# EPICS StreamDevice protocol: visarCameraApp/srcProtocol/visar.proto
################################################
#                                              #
#  Stream Protocol File for the Visar camera   #
#                                              #
#                                              #
################################################

OutTerminator =  CR;
ReplyTimeout  =  300;
ReadTimeout   =  100;
WriteTimeout  =  100;
LockTimeout   =  300;

###############################################
#  Camera Parameters                          #
###############################################

#########################################
#  Exposure time                        #
#########################################

set_exposure_time{
    InTerminator = ;
    ExtraInput   = Ignore;
	out "CamParamSet(Live,Exposure,%.6f %(\$1AcquireTimeVisarUnits){us|ms|s|min})";
	in "%*/(?m)0,CamParamSet\r/";
}

set_exposure_time_s{
    InTerminator = ;
    ExtraInput   = Ignore;
	out "CamParamSet(Live,Exposure,%(\$1AcquireTime).6f s)";
	in "%*/(?m)0,CamParamSet\r/";
}

get_exposure_time{
    InTerminator = ;
    ExtraInput   = Ignore;
	out "CamParamGet(Live,Exposure)";
	in  "%*/(?m)0,CamParamGet,/%f %(\$1AcquireTimeVisarUnits_RBV){us|ms|s|m}\r";
}

#########################################
#  Gain                                 #
#########################################

# II Gain / AD Gain
set_II_gain{
    InTerminator = ;
    ExtraInput   = Ignore;
	out "DevParamSet(TD,II-Gain,%d)";
	in "%*/(?m)0,DevParamSet\r/";
}

get_II_gain{
    InTerminator = "";
    ExtraInput   = Ignore;
    out "DevParamGet(TD,II-Gain)";
#	in  "%*/(.?)\r/0,DevParamGet,%s\r%*/(.?)\r";
	in "%.2/([WF].*\r)*0,DevParamGet,([0-9]+)/"
}

#########################################
#  Trigger Mode                         #
#########################################

set_mode{
    InTerminator = ;
    ExtraInput   = Ignore;
	out "DevParamSet(TD,Mode,%{Focus|Operate})";
	in "%*/(?m)0,DevParamSet\r/";
}

get_mode{
    InTerminator = ;
    ExtraInput   = Ignore;
	out "DevParamGet(TD,Mode)";
	in "%*/(?m)0,DevParamGet,/%{Focus|Operate}\r";
}

#########################################
#  Gate Mode                            #
#########################################

set_gate_mode{
    InTerminator = ;
    ExtraInput   = Ignore;
	out "DevParamSet(TD,Gate Mode,%{Normal|Gate|Open Fixed})";
	in "%*/(?m)0,DevParamSet\r/";
}

get_gate_mode{
    InTerminator = ;
    ExtraInput   = Ignore;
	out "DevParamGet(TD,Gate Mode)";
	in "%*/(?m)0,DevParamGet,/%{Normal|Gate|Open Fixed}\r";
}

#########################################
#  Shutter                              #
#########################################

set_shutter{
    InTerminator = ;
    ExtraInput   = Ignore;
	out "DevParamSet(TD,Shutter,%{Closed|Open})";
	in "%*/(?m)0,DevParamSet\r/";
}
get_shutter{
    InTerminator = ;
    ExtraInput   = Ignore;
	out "DevParamGet(TD,Shutter)";
	in "%*/(?m)0,DevParamGet,/%{Closed|Open}\r";
}

#########################################
#  Image Mode                           #
#########################################

set_image_mode{
    InTerminator = ;
    ExtraInput   = Ignore;
	out "DevParamSet(TD,Trig. Mode,%{Single|Cont|Cont})";
	in "%*/(?m)0,DevParamSet\r/";
}
get_image_mode{
    InTerminator = ;
    ExtraInput   = Ignore;
	out "DevParamGet(TD,Trig. Mode)";
	in "%*/(?m)0,DevParamGet,/%{Single|Cont|xx}\r";
}

#########################################
#  Trigger Status                       #
#########################################

set_trigger_status{
    InTerminator = ;
    ExtraInput   = Ignore;
	out "DevParamSet(TD,Trigger status,%{Ready|Fired|Do Reset})";
	in "%*/(?m)0,DevParamSet\r/";
}

get_trigger_status{
    InTerminator = ;
    ExtraInput   = Ignore;
	out "DevParamGet(TD,Trigger status)";
	in "%*/(?m)0,DevParamGet,/%{Ready|Fired|Do Reset}\r";
}

#########################################
#  Time Range                           #
#########################################

set_time_range{
    InTerminator = ;
    ExtraInput   = Ignore;
	out "DevParamSet(TD,Time Range,%{0.5 ns|1 ns|2 ns|5 ns|10 ns|20 ns|50 ns|100 ns|200 ns|500 ns|1 us|2 us|5 us|10 us|20 us|50 us})";
	in "%*/(?m)0,DevParamSet\r/";
}

get_time_range{
    InTerminator = ;
    ExtraInput   = Ignore;
	out "DevParamGet(TD,Time Range)";
	in "%*/(?m)0,DevParamGet,/%{0.5 ns|1 ns|2 ns|5 ns|10 ns|20 ns|50 ns|100 ns|200 ns|500 ns|1 us|2 us|5 us|10 us|20 us|50 us}\r";
}

#########################################
#  Focus Time Over                      #
#########################################

set_focus_time_over{
    InTerminator = ;
    ExtraInput   = Ignore;
    out "DevParamSet(TD,FocusTimeOver,%d)";
    in "%*/(?m)0,DevParamSet\r/";
}

get_focus_time_over{
    InTerminator = ;
    ExtraInput   = Ignore;
   out "DevParamGet(TD,FocusTimeOver)";
   in "%*/(?m)0,DevParamGet,/%d\r";
}

###############################################
#  Camera Parameters                          #
###############################################

#########################################
#  Frame Notification                   #
#########################################

buffer_notification{
    LockTimeout = 100;
    ReplyTimeout = 100;
    ReadTimeout = 100;
    InTerminator = CR;
    in "4,Livemonitor,RingBuffer,%d";
}

#########################################
#  Frame Rate notification              #
#########################################

frame_rate_notification{
    LockTimeout = 100;
    ReplyTimeout = 100;
    ReadTimeout = 100;
    InTerminator = CR;
    in "4,Frame rate %f Hz";
}

#########################################
#  Generic notification     #
#########################################

generic_notification{
    LockTimeout = 100;
    ReplyTimeout = 100;
    ReadTimeout = 100;
    InTerminator = CR;
    in "4,%s";
}

###############################################
#  Commands                                   #
###############################################

#########################################
#  Get Frame                            #
#########################################

get_frame{
   out "ImgDataGet(Current,Data)";
}

#########################################
#  Start capture                        #
#########################################

start_capture{
    out "AcqLiveMonitor(RingBuffer,10)";
    out "AcqStart(Live)";
}

#########################################
#  Stop Capture                         #
#########################################

stop_capture{
   out "AcqStop()";
}

#visar.proto

#########################################
#  Open Application                     #
#########################################

start_app{
    out "AppStart()";
}

#########################################
#  Close Application                    #
#########################################

stop_app{
    out "AppEnd()";
}
